FUNCTION TryConvert_LREAL_TO_TIME : BOOL
VAR_INPUT
	in : LREAL;
	out : REFERENCE TO TIME;
END_VAR

IF in > DatatypeLimits.MAX_VALUE_OF_LREAL_WHICH_CAN_BE_HELD_IN_A_TIME THEN
	RETURN;
END_IF

IF in < DatatypeLimits.MIN_VALUE_OF_LREAL_WHICH_CAN_BE_HELD_IN_A_TIME THEN
	RETURN;
END_IF

out := LREAL_TO_TIME(in);
TryConvert_LREAL_TO_TIME := TRUE;

END_FUNCTION

(* stored: Version 1.1.0.1, ProductVersion 3.1.4024.12
   POU TryConvert_LREAL_TO_TIME: Id {a51c627c-ff96-4002-9c37-c07f80ed2784}, SpecialFunc None *)
